// Mitsubishi GX Works2 project: 0702-4   PLC: Q02/Q02H

PROGRAM MAIN
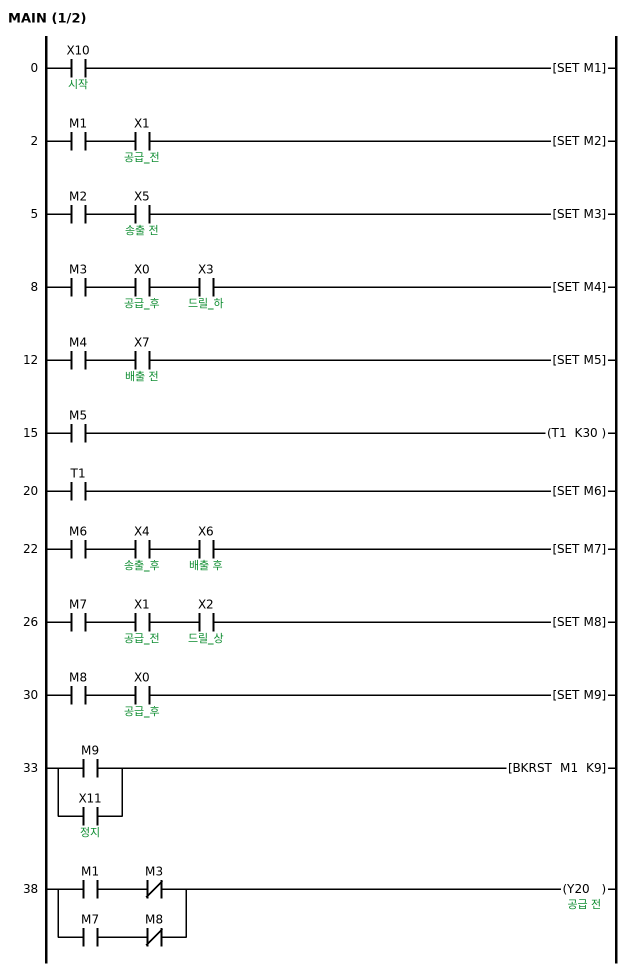
0     LD      X10  ; 시작
      SET     M1
2     LD      M1
      AND     X1  ; 공급_전
      SET     M2
5     LD      M2
      AND     X5  ; 송출 전
      SET     M3
8     LD      M3
      AND     X0  ; 공급_후
      AND     X3  ; 드릴_하
      SET     M4
12    LD      M4
      AND     X7  ; 배출 전
      SET     M5
15    LD      M5
      OUT     T1 K30
20    LD      T1
      SET     M6
22    LD      M6
      AND     X4  ; 송출_후
      AND     X6  ; 배출 후
      SET     M7
26    LD      M7
      AND     X1  ; 공급_전
      AND     X2  ; 드릴_상
      SET     M8
30    LD      M8
      AND     X0  ; 공급_후
      SET     M9
33    LD      M9
      OR      X11  ; 정지
      BKRST   M1 K9
38    LD      M1
      ANI     M3
      LD      M7
      ANI     M8
      ORB
      OUT     Y20  ; 공급 전
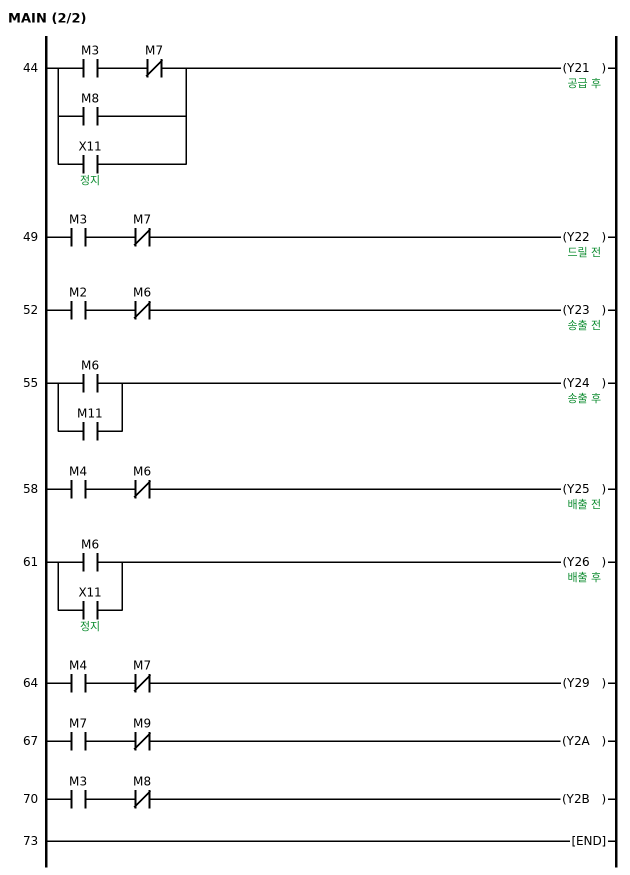
44    LD      M3
      ANI     M7
      OR      M8
      OR      X11  ; 정지
      OUT     Y21  ; 공급 후
49    LD      M3
      ANI     M7
      OUT     Y22  ; 드릴 전
52    LD      M2
      ANI     M6
      OUT     Y23  ; 송출 전
55    LD      M6
      OR      M11
      OUT     Y24  ; 송출 후
58    LD      M4
      ANI     M6
      OUT     Y25  ; 배출 전
61    LD      M6
      OR      X11  ; 정지
      OUT     Y26  ; 배출 후
64    LD      M4
      ANI     M7
      OUT     Y29
67    LD      M7
      ANI     M9
      OUT     Y2A
70    LD      M3
      ANI     M8
      OUT     Y2B
73    END
END_PROGRAM
